{attribute 'GeneratedUsingTerminal: EL6201-0000-0017'}
{attribute addProperty BoxType "EL6201-0000-0017"}
{attribute addProperty Id "Slave_24A_DI0BOOL1Slave_24A_DI1BOOL1Slave_24A_DI2BOOL1Slave_24A_DI3BOOL1Slave_24B_DI0BOOL1Slave_24B_DI1BOOL1Slave_24B_DI2BOOL1Slave_24B_DI3BOOL1"}
{attribute addProperty CRC "3569941483"}
{attribute addProperty Size "8"}
TYPE Slave_24_Inputs_D4C8FBEB :
STRUCT
	{attribute addProperty Name "Slave_24A_DI0"}
	Slave_24A_DI0 : BOOL;
	{attribute addProperty Name "Slave_24A_DI1"}
	Slave_24A_DI1 : BOOL;
	{attribute addProperty Name "Slave_24A_DI2"}
	Slave_24A_DI2 : BOOL;
	{attribute addProperty Name "Slave_24A_DI3"}
	Slave_24A_DI3 : BOOL;
	{attribute addProperty Name "Slave_24B_DI0"}
	Slave_24B_DI0 : BOOL;
	{attribute addProperty Name "Slave_24B_DI1"}
	Slave_24B_DI1 : BOOL;
	{attribute addProperty Name "Slave_24B_DI2"}
	Slave_24B_DI2 : BOOL;
	{attribute addProperty Name "Slave_24B_DI3"}
	Slave_24B_DI3 : BOOL;
END_STRUCT
END_TYPE

(* stored: Version 1.2.0.0, ProductVersion 3.1.4024.9
   DUT Slave_24_Inputs_D4C8FBEB: Id {1226c8b7-fc6e-4850-87ad-4b01a511930e} *)
